FUNCTION_BLOCK FB_PTM_Agilent_NoFeedback EXTENDS FB_Pump
VAR_INPUT
    i_xExtILKOk : BOOL; // Connect to external interlock logic(e.g TURBO_ILK Function), TRUE if not used.
    i_stGauge	:	ST_VG; //Pirani backing gauge for pump interlock
    i_rMaxBackingPressure : REAL;
END_VAR
VAR_OUTPUT
    {attribute 'pytmc' :=' pv:'}
    iq_stPtm	:	ST_AgilentPTM;
END_VAR
VAR
    {attribute 'instance-path'}
    {attribute 'noinit'}
    sPath: STRING;
    //xRunOk	:	BOOL;
    nMaxR1Fault: INT :=5;
    nR1Fault : INT;
    tFaultWindowDuration : TIME := T#300S;
    tR1FaultDuration : TIME := T#120S;
    tTimeOutDuration: TIME:= T#10M;
    tFaultWindowElapsed: TON;
    tR1Fault : TON;
    tStartTimeOut : TON;
    tR1TimeOut: TON;
    step : INT :=0;
    nErrorCode: INT :=0;
    xBackingPressureOK: BOOL;
    iMaxSpeed : INT:=963;

    rPowerScale: REAL:=10;//W
    rCurrentScale: REAL:=1;//A

    (*I/Os*)
    i_xSTART 	AT%I*:	BOOL;
    i_xR1	AT%I*	:  BOOL;
    i_xR2	AT%I*	:  BOOL;
    i_xLSpd	AT%I*:  BOOL;
    i_iTempMon AT%I*: INT;
    i_iPowerMon AT%I*: INT;
    i_iCurrentMon AT%I*: INT;
    i_iRawSpeed AT %I* : INT;
    i_xFault AT%I*	:	BOOL;
    q_RunDO AT%Q*	:	BOOL;
    q_xLSpd	AT%Q*	:  BOOL;


    // For logging
  //  Msg : FB_FormatString;
   // fbJson : FB_JsonSaxWriter;
   tOverrideActivated : R_TRIG;

    iTermBits: UINT := 32767 ; // The terminal's maximum value in bits
END_VAR

(* Basic Agilent Turbo Controls *)
(* Allen Pai, 2021-02-02 *)

(*FB_Input Link ingto Data Structure*)
iq_stPtm.xExtRunOk := i_xExtILKOk;
(*Validate Backing Pressure set point doesn't exceed the Maximum backingPressure*)
iq_stPtm.rBackingPressureSP := BackingPressureSetPoint(iq_stPtm.rBackingPressureSP,i_rMaxBackingPressure);

(* state machine *)
CASE (step) OF
(*Pump Stopped State*)
    0: // Pump Stopped State
        iq_stPtm.xRunSW:=FALSE;
        //Reset Output signals;
        iq_stPtm.q_RunDO:=FALSE;
        iq_stPtm.q_xSS := FALSE;
        iq_stPtm.q_xLSpd:= FALSE;
        iq_stPtm.eState := pumpSTOPPED;
        step:=10;

(*Idle State waiting to start*)
    10: // Idle State, waiting for the xRunSwitch
        IF iq_stPtm.xExtRunOk  AND iq_stPTM.xRunSW THEN
            iq_stPtm.q_RunDO := iq_stPTM.xRunSW; //
            step:=20;
        END_IF


(*Pump On State*)
    20: // Pump is On
        iq_stPtm.q_RunDO := iq_stPTM.xRunSW; // done in previous state
        //If External Interlock is false or Operator has stopped pump, turn off pump
        IF (iq_stPtm.xExtRunOk= FALSE) OR (iq_stPTM.xRunSW = FALSE) THEN
            step:= 0;
        ELSE
            step:=20;
        END_IF
END_CASE

(*Check backing gauge pressure*)
//xBackingPressureOK := i_stGauge.xPRESS_OK AND ( i_stGauge.rPRESS < iq_stPtm.rBackingPressureSP);

(* IO Mapping*)
IO();
(*Assign Error Message*)
//iq_stPtm.sError := ErrorMessage(nErrorCode, iq_stPtm.eState);
// Log States and triggers
//ACT_Logger();

ACT_Interlock();

ACTION ACT_Interlock:
This^.tILK(IN:= (i_stGauge.rPRESS>=iq_stPtm.rBackingPressureSP), PT:=T#5S, Q=> );
END_ACTION

METHOD BackingPressureSetPoint : REAL
VAR_INPUT
    i_SetPoint : REAL;
    rMaxBackingPressure: REAL;
END_VAR
BackingPressureSetPoint := Min(i_SetPoint , rMaxBackingPressure);
END_METHOD

ACTION IO:
(*inputs*)
iq_stPtm.i_xSTART:=	i_xSTART;
iq_stPtm.i_xR1:=	i_xR1;
iq_stPtm.i_xR2:=	i_xR2;
iq_stPtm.i_xLSpd:=	i_xLSpd;
iq_stPtm.i_xFault:=	i_xFault;
(* Real-value calculation *)
If (iTermBits=0) THEN iTermBits := 32767;
END_IF
(*iq_stPtm.i_rCurrentMon := (10*(i_iCurrentMon)/iTermBits)*rCurrentScale;
iq_stPtm.i_rTempMon := 10*INT_TO_REAL(i_iTempMon)/iTermBits;
iq_stPtm.i_rPowerMon := (10*INT_TO_REAL(i_iPowerMon)/iTermBits)*rPowerScale;
iq_stPtm.i_diCurSpd := 10*LREAL_TO_DINT(INT_TO_REAL(i_iRawSpeed)/iTermBits);
*)

(*outputs*)
q_RunDO := iq_stPtm.q_RunDO;
q_xLSpd := iq_stPtm.q_xLSpd;
END_ACTION

END_FUNCTION_BLOCK

(* stored: Version 1.1.0.1, ProductVersion 3.1.4022.18
   POU FB_PTM_Agilent_NoFeedback: Id {cb2eb156-7e3f-48fe-afc1-860bf870e3b3}, SpecialFunc None
   Action ACT_Interlock: Id {5e7862f2-c7a8-4e45-afd4-ac1a5f6a4ad4}
   Method BackingPressureSetPoint: Id {167982aa-a2b8-40d9-9c64-b30de296433b}
   Action IO: Id {2f6d0b8a-91f1-4e9e-a012-c189d0d51d98} *)
